FUNCTION_BLOCK FB_Blinker
VAR_INPUT
END_VAR
VAR_OUTPUT
END_VAR
VAR
END_VAR

END_FUNCTION_BLOCK

(* stored: Version 1.1.0.1, ProductVersion 3.1.4024.11
   POU FB_Blinker: Id {728443ba-9c90-46c1-b845-e3ce5de893a2}, SpecialFunc None *)
